# EPICS autosave request: GalilSup/Db/galil_8_motor_extras.req
file "galil_motor_extras.req",  P=$(P), M=$(M1)
file "galil_motor_extras.req",  P=$(P), M=$(M2)
file "galil_motor_extras.req",  P=$(P), M=$(M3)
file "galil_motor_extras.req",  P=$(P), M=$(M4)
file "galil_motor_extras.req",  P=$(P), M=$(M5)
file "galil_motor_extras.req",  P=$(P), M=$(M6)
file "galil_motor_extras.req",  P=$(P), M=$(M7)
file "galil_motor_extras.req",  P=$(P), M=$(M8)
